Fanuc KAREL source: CNV_TIME_STR.kl

PROGRAM T
%NOLOCKGROUP
VAR
 v0 : INTEGER
 v1 : STRING[40]
BEGIN
 CNV_TIME_STR(v0, v1)
END T
